TYPE ST_OutputsSickScanner :
STRUCT	
	ConfMessageOut			: ARRAY[0..31] OF BYTE;	
	Trigger					: BOOL;		//Trigger signal to scanner -> Start scan and keep scan while trigger is set or barcode is read.
END_STRUCT
END_TYPE

(* stored: Version 1.1.0.1, ProductVersion 3.1.4024.4
   DUT ST_OutputsSickScanner: Id {85ff9338-8983-44f4-a60f-b8e19f769c67} *)
